Omron CX-Programmer project NewProject (CX-Programmer 9.75)

# PLC TrafficLight: CP1E N30

## Program NewProgram1 (cyclic task 0)
Local symbols
Green 100.03 BOOL
MainSupply 100.00 BOOL
Red 100.01 BOOL
Start 0.00 BOOL
Stop 0.01 BOOL
Sw1 0.02 BOOL
Sw2 0.03 BOOL
Sw3 0.04 BOOL
Yellow 100.02 BOOL

### Section Section1

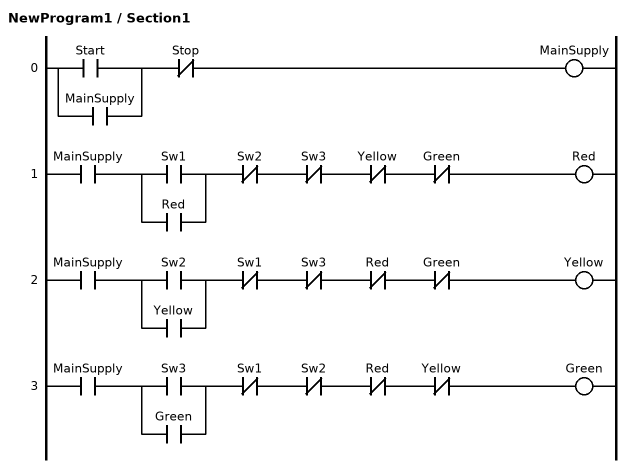
; rung 0
LD Start
OR MainSupply
ANDNOT Stop
OUT MainSupply
; rung 1
LD MainSupply
LD Sw1
OR Red
ANDLD
ANDNOT Sw2
ANDNOT Sw3
ANDNOT Yellow
ANDNOT Green
OUT Red
; rung 2
LD MainSupply
LD Sw2
OR Yellow
ANDLD
ANDNOT Sw1
ANDNOT Sw3
ANDNOT Red
ANDNOT Green
OUT Yellow
; rung 3
LD MainSupply
LD Sw3
OR Green
ANDLD
ANDNOT Sw1
ANDNOT Sw2
ANDNOT Red
ANDNOT Yellow
OUT Green

### Section END
; rung 0
END(001)